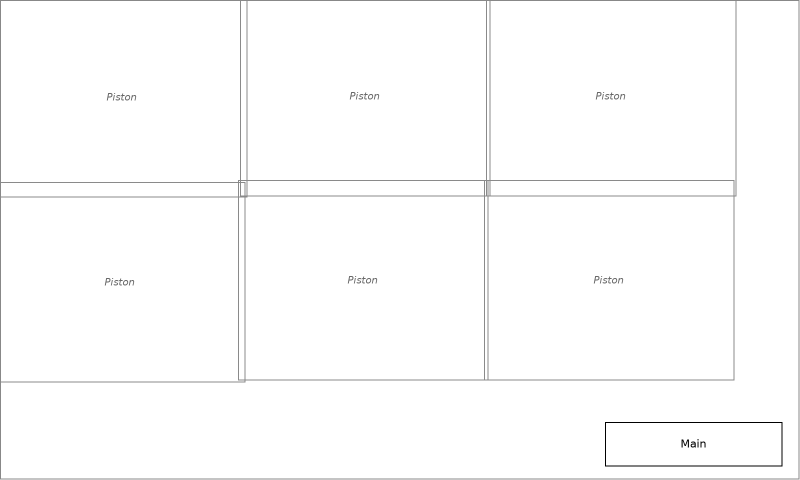
VISUALIZATION PistonsManual  // 800x480
    Frame (-3,-3 250x200)
        shows Piston(piston := GVL_HMI.stSepSol1)
    Rectangle (605,422 177x44), "Main"
        OnMouseDown: change screen: Main
    Frame (-5,182 250x200)
        shows Piston(piston := GVL_HMI.stPushSol1)
    Frame (240,-4 250x200)
        shows Piston(piston := GVL_HMI.stSepSol2)
    Frame (238,180 250x200)
        shows Piston(piston := GVL_HMI.stPushSol2)
    Frame (486,-4 250x200)
        shows Piston(piston := GVL_HMI.stSepSol3)
    Frame (484,180 250x200)
        shows Piston(piston := GVL_HMI.stPushSol3)
END_VISUALIZATION

(* stored: Version 1.1.0.1, ProductVersion 3.1.4024.16
   Visu PistonsManual: Id {5acef5c4-26de-424a-ba91-a13d601f943c} *)
